PROGRAM MAIN
VAR
	sensor1 : BOOL;
	sensor2 : BOOL;
	sensor3 : BOOL;
	counter1 : INT;
	
	seq : Sequencer;
	firstCycle : BOOL := TRUE;
	test : BOOL;
	ceres : CResult;
	n1 : PVOID;
	n2 : PVOID;
	n3 : PVOID;
	
	re : Regex;
END_VAR

IF firstCycle THEN
	firstCycle := FALSE;
	
	RegisterActions();
	
END_IF

seq();

CASE seq.currentAction.caseNumber OF
	0 : // action code 1
	10 : // action code 2
	20 : // action code 3
	30 : // action code 4

END_CASE

Is(test);
Is(ceres);

n1 := SIZEOF(CResult);
n2 := SIZEOF(CResult.result);
n3 := SIZEOF(CResult.datatype);

re.match(pattern := 'he.*o', text := 'hellQQllo_HelloWorld').found;

ACTION RegisterActions:
//seq.ClearActions();

//seq.RegisterAction(
//	name := 'name 1',
//	number := 0
//);
//seq.RegisterAction(
//	name := 'name 2',
//	number := 10
//);
//seq.RegisterAction(
//	name := 'name 3',
//	number := 20
//);
//seq.RegisterAction(
//	name := 'name 4',
//	number := 30
//);
END_ACTION

ACTION RegisterAll:
// Register actions
seq.RegisterAction(
	name := 'name 1',
	caseNumber := 0,
	''
);
seq.RegisterAction(
	name := 'name 2',
	caseNumber := 10,
	''
);
seq.RegisterAction(
	name := 'name 3',
	caseNumber := 20,
	''
);
seq.RegisterAction(
	name := 'name 4',
	caseNumber := 30,
	''
);

// Register conditions
seq.RegisterCondition('cond 1').Is(sensor1);
seq.RegisterCondition('cond 2').Is(sensor2).AndIs(sensor3);
seq.RegisterCondition('cond 3').Is(sensor3);
seq.RegisterCondition('cond 4').Is(sensor3);

// Bind them together
seq.Bind('name 1')
	.WhenGoTo('cond 1', 'name 2');
seq.Bind('name 2')
	.WhenGoTo('cond 2', 'name 3')
	.WhenGoTo('cond 3', 'name 4');
seq.Bind('name 3')
	.WhenGoTo('cond 3', 'name 4');
seq.Bind('name 4')
	.WhenGoTo('cond 4', 'name 1');
END_ACTION

ACTION RegisterConditions:
//seq.ClearConditions();

//seq.RegisterCondition('cond 1').Is(sensor1);
//seq.RegisterCondition('cond 2').Is(sensor2).AndIs(sensor3);
//seq.RegisterCondition('cond 3').Is(sensor3);
//seq.RegisterCondition('cond 4').Is(sensor3);
END_ACTION

ACTION RegisterTransitions:
//seq.Bind('name 1')
//	.WhenGoTo('cond 1', 'name 2');
//seq.Bind('name 2')
//	.WhenGoTo('cond 2', 'name 3')
//	.WhenGoTo('cond 3', 'name 4');
//seq.Bind('name 3')
//	.WhenGoTo('cond 3', 'name 4');
//seq.Bind('name 4')
//	.WhenGoTo('cond 4', 'name 1');
END_ACTION

END_PROGRAM

(* stored: Version 1.1.0.1, ProductVersion 3.1.4024.11
   POU MAIN: Id {711c9c87-dd2c-40bf-a050-a3708e521dd8}, SpecialFunc None
   Action RegisterActions: Id {663b0111-1fee-4952-b388-ee530e3b0e65}
   Action RegisterAll: Id {d88f312f-a0ad-4b5d-93e2-81141268fc29}
   Action RegisterConditions: Id {ee97d2a6-ceaa-455d-8101-7fa903610d86}
   Action RegisterTransitions: Id {c8a3c281-1247-4144-bb87-275feaa83da2} *)
